FUNCTION_BLOCK FB_HMI_DETECTORS EXTENDS FB_HMI_COMPONENT
VAR_INPUT
END_VAR
VAR_OUTPUT
END_VAR
VAR
END_VAR

END_FUNCTION_BLOCK

(* stored: Version 1.1.0.1, ProductVersion 3.1.4024.14
   POU FB_HMI_DETECTORS: Id {bb010f4b-1000-4749-99c5-3feb9c8a669c}, SpecialFunc None *)
